(* CODESYS project Cilindros.project
   Title: Sin título
   Version: 0.0.0.0
   Author: serbogr1

Project tree, tasks and I/O mapping:
  MyController : TM241CE40R, Schneider Electric, order no. TM241CE40R, version 4.0.6.18
    application Application
      task MAST (cyclic, interval 20 ms, priority 15, watchdog 100 ms x 1) calls My_Main, Secuencia
      global variables GVL
      program My_Main [SFC]
      visualisation My_Visu
      program Secuencia [SFC]
    DI : Digital Inputs, Schneider Electric, version 4.0.6.18
        input  idwDI_IDW0 : DWORD  // IDW0
        input  ibDI_IB1 : BYTE  // IB1
    DQ : Digital Outputs, Schneider Electric, version 4.0.6.18
        output qwDQ_QW0 : WORD  // QW0
        output qbDQ_QB1 : BYTE  // QB1
    Counters : Counters, Schneider Electric, version 4.0.6.18
    Pulse_Generators : Pulse Generators, Schneider Electric, version 4.0.6.18
    Cartridge_1 : Cartridge, Schneider Electric, version 4.0.6.18
    Cartridge_2 : Cartridge, Schneider Electric, version 4.0.6.18
    IO_Bus : IO bus - TM3, Schneider Electric, version 4.0.6.18
    COM_Bus : COM bus, Schneider Electric, version 4.0.6.18
    Ethernet_1 : Ethernet Network, Schneider Electric, version 4.0.6.18
        settings: WebServer = TRUE; FTP Server = TRUE; SoMachine Protocol = TRUE; Modbus Server = TRUE; NetManage Protocol = TRUE; SNMP protocol = TRUE; Enable Routing = FALSE; WebVisu protocol = TRUE; DHCP Server Active = FALSE
    Serial_Line_1 : Serial line, Schneider Electric, version 4.0.6.18
      SoMachine_Network_Manager : SoMachine-Network Manager, Schneider Electric, version 4.0.0.2
    Serial_Line_2 : Serial line, Schneider Electric, version 4.0.6.18
      Modbus_Manager : Modbus Manager, Schneider Electric, version 4.0.0.2
  text list GlobalTextList
*)

// MyController/Application/GVL
VAR_GLOBAL
END_VAR
VAR_GLOBAL
	BP_Verde: BOOL;
	BP_Negro: BOOL;
	BS2P_DE: BOOL;
	BS3P_I_IZ: BOOL;
	BS3P_II_DE: BOOL;
	SETA: BOOL;
	CSS_FUERA AT %IX0.6: BOOL;
	CCS_FUERA AT %IX0.7: BOOL;
	CCS_DENTRO AT %IX1.0: BOOL;
	CIS_FUERA AT %IX1.1: BOOL;
	PINZA_ABIERTA AT %IX1.2: BOOL;
	PINZA_CERRADA AT %IX1.3: BOOL;
	CR_INICIO AT %IX1.4: BOOL;
	CR_FINAL AT %IX1.5: BOOL;
	SUCCION AT %IX1.6: BOOL;
	VENTOSA AT %IX1.7: BOOL;
	SACAR_CS AT %QX0.4: BOOL;
	SACAR_CC AT %QX0.5: BOOL;
	INTRODUCIR_CC AT %QX0.6: BOOL;
	SACAR_CI AT %QX0.7: BOOL;
	CERRAR_PINZA AT %QX1.0: BOOL;
	ABRIR_PINZA AT %QX1.1: BOOL;
	CR_HORARIO AT %QX1.2: BOOL;
	VACIO_VENTOSA AT %QX1.3: BOOL;
	B_PILOTO_V AT %QX1.4: BOOL;
	B_PILOTO_B AT %QX1.5: BOOL;
	B_PILOTO_R AT %QX1.6: BOOL;
END_VAR

// MyController/Application/My_Main
PROGRAM My_Main
VAR
END_VAR

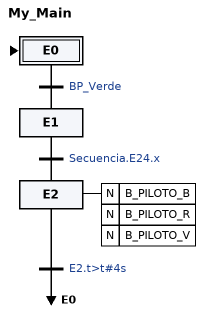
INITIAL_STEP E0:
END_STEP
TRANSITION FROM E0 TO E1
    := BP_Verde;
END_TRANSITION
STEP E1:
END_STEP
TRANSITION FROM E1 TO E2
    := Secuencia.E24.x;
END_TRANSITION
STEP E2:
    B_PILOTO_B(N);
    B_PILOTO_R(N);
    B_PILOTO_V(N);
END_STEP
TRANSITION FROM E2 TO E0
    := E2.t>t#4s;
END_TRANSITION

END_PROGRAM

// MyController/Application/Secuencia
PROGRAM Secuencia

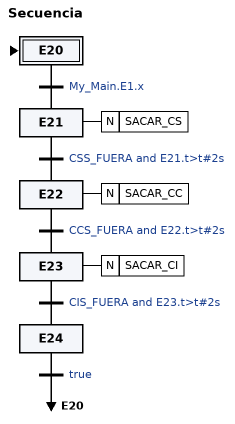
INITIAL_STEP E20:
END_STEP
TRANSITION FROM E20 TO E21
    := My_Main.E1.x;
END_TRANSITION
STEP E21:
    SACAR_CS(N);
END_STEP
TRANSITION FROM E21 TO E22
    := CSS_FUERA and E21.t>t#2s;
END_TRANSITION
STEP E22:
    SACAR_CC(N);
END_STEP
TRANSITION FROM E22 TO E23
    := CCS_FUERA and E22.t>t#2s;
END_TRANSITION
STEP E23:
    SACAR_CI(N);
END_STEP
TRANSITION FROM E23 TO E24
    := CIS_FUERA and E23.t>t#2s;
END_TRANSITION
STEP E24:
END_STEP
TRANSITION FROM E24 TO E20
    := true;
END_TRANSITION

END_PROGRAM

// MyController/Application/My_Visu
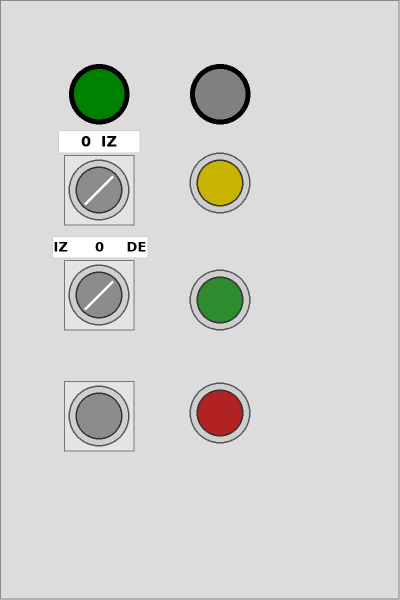
VISUALIZATION My_Visu  // 400x600, background image 
    Lamp1 (185,265 70x70), variable: B_PILOTO_V, style: Lamp-Lamp1-Green
    Lamp1 (185,148 70x70), variable: B_PILOTO_B, style: Lamp-Lamp1-Yellow
    Lamp1 (185,378 70x70), variable: B_PILOTO_R, style: Lamp-Lamp1-Red
    RotarySwitch (64,155 70x70), behaviour: TOGGLE, style: Switch-RotarySwitch-Gray
    Ellipse (69,64 60x60), colour toggle: BP_Verde
        tap BP_Verde
    Ellipse (190,64 60x60), colour toggle: BP_Verde
        tap BP_Negro
    PushSwitchLed (64,381 70x70), behaviour: TOGGLE, style: Switch-PushSwitchLed-Gray
    RotarySwitch (64,260 70x70), behaviour: TOGGLE, style: Switch-RotarySwitch-Gray
    Textfield (58,130 82x23), "0 IZ"
    Textfield (52,236 96x22), "IZ 0 DE"
END_VISUALIZATION
